// Returns the datatype of a variable as a string using its path.
FUNCTION FsF_GetTypeNameByPath : FsT_Str
VAR_INPUT
	Path : FsT_LStr; // Variable/Symbol path as string | e.g. 'MAIN.nVar'
END_VAR
VAR 
	nTmp : UDINT := SIZEOF(FsF_GetTypeNameByPath);
END_VAR

FsF_IecApplicationInformation().GetSymbolDatatype(Path, nTmp, ADR(FsF_GetTypeNameByPath));

END_FUNCTION

(* stored: Version 1.1.0.1, ProductVersion 3.1.4024.4
   POU FsF_GetTypeNameByPath: Id {b78d29b7-a201-4bb0-8581-654cfe213643}, SpecialFunc None *)
